// TIA Portal V16 export
// export: Created 2021-11-12T13:31:58.4175263Z, ExportSetting WithDefaults, DisplayName Totally Integrated Automation Portal, DisplayVersion V16 Update 3, DisplayName TIA Portal Version Control Interface, DisplayVersion V16 Update 2, DisplayName TIA Portal Openness, DisplayVersion V16 Update 3, DisplayName SINAMICS Startdrive Advanced, DisplayVersion V16 Update 5, DisplayName SINAMICS Startdrive G130, G150, S120, S150, SINAMICS MV, S210, DisplayVersion V16 Update 5, DisplayName SINAMICS Startdrive G110M, G120, G120C, G120D, G120P, G115D, DisplayVersion V16 Update 5, DisplayName STEP 7 Professional, DisplayVersion V16 Update 3, DisplayName STEP 7 Safety, DisplayVersion V16, DisplayName WinCC UA Professional, DisplayVersion V16 Update 3
DATA_BLOCK "IDB_Zone000"   // DB177
VERSION : 0.1
// stored: AutoNumber true, DBAccessibleFromOPCUA true, InstanceOfName Zone000, InstanceOfType FB
"Zone000"
   // VAR
   //    SF_StationMEM1Mode { S7_SetPoint := 'True'} : "STD_Station";
   //    "SF_EQ01-MA01" : "STD_Drive1";
   //    "SF_EQ01-MA02" : "STD_Drive1";
   //    "SF_EQ02-MA01" : "STD_Drive1";
   //    "SF_UC11-TA01" { S7_SetPoint := 'True'} : "STD_Siemens_G120_CU240E_2_PN";
   //    "SF_UC11-TA02" { S7_SetPoint := 'True'} : "STD_Siemens_G120_CU240E_2_PN";
   //    "SF_UC11-TA03" { S7_SetPoint := 'True'} : "STD_Siemens_G120_CU240E_2_PN";
   //    SS_Edge { S7_SetPoint := 'True'} : Array[0..100] of Bool;
   //    SB1_PowerOk { S7_SetPoint := 'True'} : Bool;
   // END_VAR
BEGIN
END_DATA_BLOCK
